TEXTLIST TL_Params_Enum
  1 = 'OutputSel_H'
  2 = 'OutputSel_C'
  3 = 'TempSensTerm'
  4 = 'SensorType'
  5 = '*** not Used ***'
  6 = '*** not Used ***'
  7 = '*** not Used ***'
  8 = '*** not Used ***'
  9 = '*** not Used ***'
   = ''
END_TEXTLIST

(* stored: Version 1.1.0.1, ProductVersion 3.1.4020.12
   TextList TL_Params_Enum: Id {4a9e1b26-0421-4f99-a47b-5adc71328173} *)
